// TwinCAT 3 PLC project E_StructuredLogging
// ProgramVersion: 3.1.4023.0
// libraries:
//   log4TC, * (mbc engineering GmbH)
//   Tc2_Standard, * (Beckhoff Automation GmbH)
//   Tc2_System, * (Beckhoff Automation GmbH)
//   Tc3_Module, * (Beckhoff Automation GmbH)
// project tree:
//   / MAIN.TcPOU, PlcTask.TcTTO
// (motion and I/O tree: see PLC project a_simplelogmessage)
// real-time tasks:
//   TASK PlcTask: cycle T#10ms, priority 20, ADS port 350
//   TASK PlcTask1: cycle T#10ms, priority 21, ADS port 351
//   TASK PlcTask2: cycle T#10ms, priority 22, ADS port 352

CONFIGURATION E_StructuredLogging
    RESOURCE PLC ON TwinCAT3
        TASK PlcTask(INTERVAL := T#10ms, PRIORITY := 20);
        PROGRAM MAIN WITH PlcTask : MAIN;
    END_RESOURCE
END_CONFIGURATION

// ---- MAIN.TcPOU
PROGRAM MAIN
VAR CONSTANT
	sLogger		: STRING := 'MAIN';
END_VAR
VAR
	nCounter	: UINT;
	fbCountTime	: TON := (PT:=T#1S);
	fTemp		: REAL := 22.3;
	fPrevTemp	: REAL;
END_VAR

IF _TaskInfo[GETCURTASKINDEXEX()].FirstCycle THEN
	F_LogL(E_LogLevel.eInfo, sLogger, 'SPS Task gestartet.');
END_IF

fbCountTime(IN:=NOT fbCountTime.Q);
IF fbCountTime.Q THEN
	nCounter := nCounter + 1;
	F_LogLA1C(
		E_LogLevel.eDebug, 
		sLogger, 
		'Zähler geändert, neuer Wert {0}', 
		nCounter, 
		F_LogContext().AddInt('MachineNo', 42)
	);
END_IF

IF fTemp <> fPrevTemp THEN
	fPrevTemp := fTemp;
	
	F_LogLA1C(
		E_LogLevel.eInfo, 
		sLogger, 
		'Temperatur {temperature}', 
		fTemp, 
		F_LogContext().AddBool('csv', TRUE)
	);
END_IF

PRG_TaskLog.Call();

END_PROGRAM
